Yaskawa INFORM job: WELDING-BACK-ST-1.JBI

/JOB
//NAME WELDING-BACK-ST-1
//POS
///NPOS 0,0,0,0,0,0
//INST
///DATE 2018/09/27 12:58
///ATTR SC,RW
NOP
IFTHEN D005=8
	'***** CMF100
	 CALL JOB:WELDING-CMF100-ST1-BACK
ENDIF
IFTHEN D005=4
	'***** F........ sensors
	 CALL JOB:WELDING-F-SENSORS-BACK-ST1
ENDIF
END
